(* Logix 5000 project; controller STAT 1756-L72 rev 20.12; software revision 20.04; part 20 of 34 *)
(* tags used below, declared in another part *)
   B14 : DINT[30];
   B17 : DINT[30];
   B3 : DINT[256];
   B9 : DINT[40];
   F8 : REAL[256];
   I19_000_Bit08 : ALIAS FOR I19[0].8;   // LACK DETECTIE NAOH
   I1_009_Bit03 : ALIAS FOR I1[9].3;   // Thermische storing pomp 1
   I1_009_Bit04 : ALIAS FOR I1[9].4;   // Pomp 1 in lijn
   I1_009_Bit07 : ALIAS FOR I1[9].7;   // Thermische storing pomp 2
   I1_009_Bit08 : ALIAS FOR I1[9].8;   // Pomp 2 in lijn
   I1_009_Bit09 : ALIAS FOR I1[9].9;   // Pomp 2 in driehoek
   I3_001_Bit15 : ALIAS FOR I3[1].15;   // Thermische storing voedingspomp fabriek 1
   I4_000_Bit00 : ALIAS FOR I4[0].0;   // Motor P3 voedingspomp in lijn
   I4_000_Bit03 : ALIAS FOR I4[0].3;   // Thermische storing voedingspomp fabriek 2
   I4_000_Bit04 : ALIAS FOR I4[0].4;   // Motor p4 in lijn in
   I6_000_Bit12 : ALIAS FOR I6[0].12;   // pressostaat osmose3
   N12 : DINT[230];
   N13 : DINT[230];
   N26 : DINT[256];
   N7 : DINT[255];
   O15_000_Bit04 : ALIAS FOR O15[0].4;   // RO3_EV1 RO3_EV1
   O15_000_Bit05 : ALIAS FOR O15[0].5;   // RO3_EV2 RO3_EV2
   T4 : TIMER[200];
(* ibt, continued *)

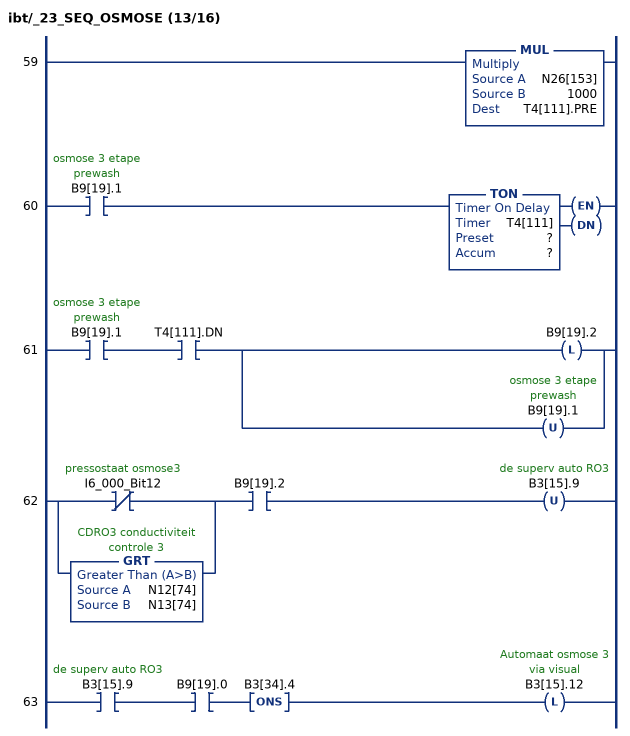
   [picture p367: ibt/_23_SEQ_OSMOSE rungs 59-63]
   59: MUL(N26[153],1000,T4[111].PRE);
   60: XIC(B9[19].1)TON(T4[111],?,?);
   61: XIC(B9[19].1)XIC(T4[111].DN)[OTL(B9[19].2) ,OTU(B9[19].1) ];
   62: [XIO(I6_000_Bit12) ,GRT(N12[74],N13[74]) ]XIC(B9[19].2)OTU(B3[15].9);
   63: XIC(B3[15].9)XIC(B9[19].0)ONS(B3[34].4)OTL(B3[15].12);
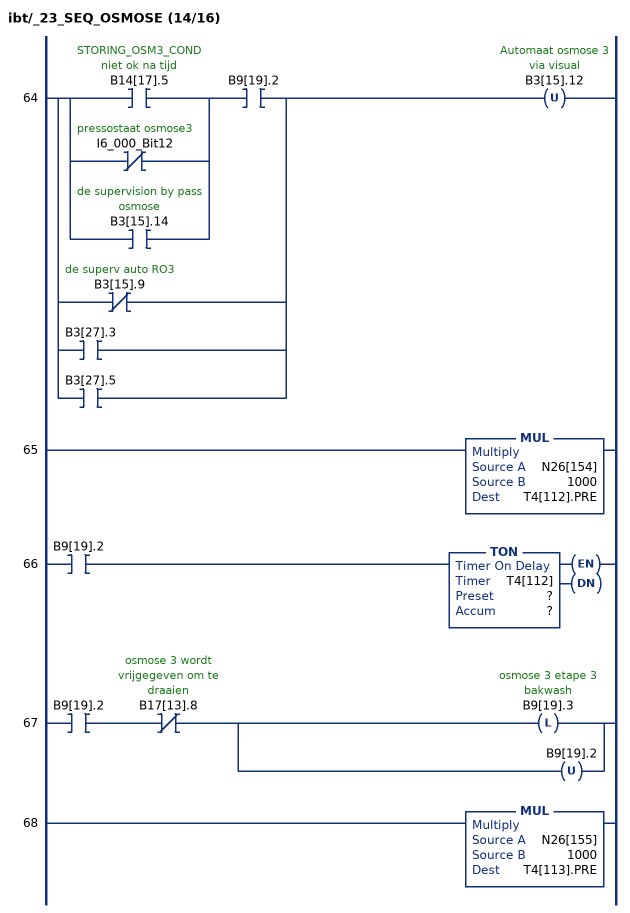
   64: [[XIC(B14[17].5) ,[XIO(I6_000_Bit12) ,XIC(B3[15].14) ] ] XIC(B9[19].2) ,XIO(B3[15].9) ,XIC(B3[27].3) ,XIC(B3[27].5) ]OTU(B3[15].12);
   65: MUL(N26[154],1000,T4[112].PRE);
   66: XIC(B9[19].2)TON(T4[112],?,?);
   67: XIC(B9[19].2)XIO(B17[13].8)[OTL(B9[19].3) ,OTU(B9[19].2) ];
   68: MUL(N26[155],1000,T4[113].PRE);
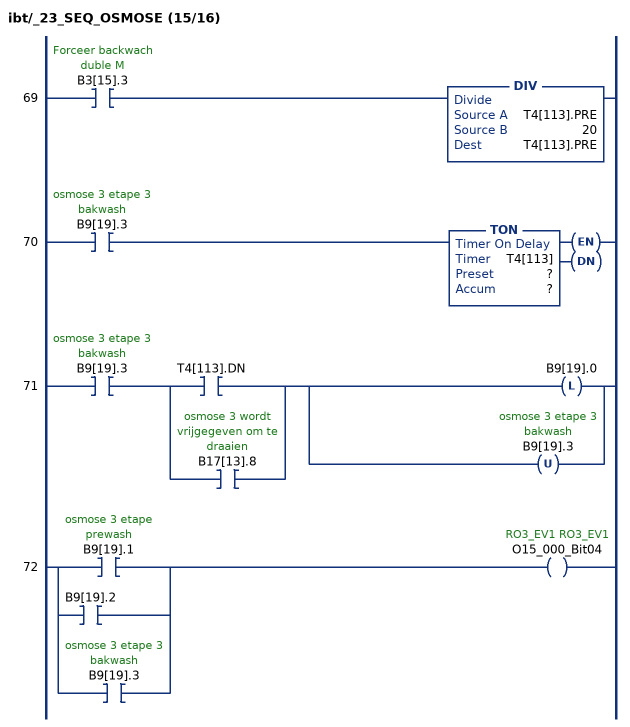
   69: XIC(B3[15].3)DIV(T4[113].PRE,20,T4[113].PRE);
   70: XIC(B9[19].3)TON(T4[113],?,?);
   71: XIC(B9[19].3)[XIC(T4[113].DN) ,XIC(B17[13].8) ][OTL(B9[19].0) ,OTU(B9[19].3) ];
   72: [XIC(B9[19].1) ,[XIC(B9[19].2) ,XIC(B9[19].3) ] ]OTE(O15_000_Bit04);
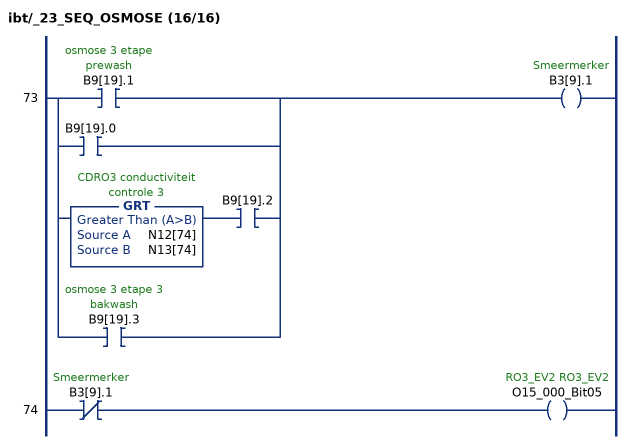
   73: [[XIC(B9[19].1) ,XIC(B9[19].0) ] ,[GRT(N12[74],N13[74]) XIC(B9[19].2) ,XIC(B9[19].3) ] ]OTE(B3[9].1);
   74: XIO(B3[9].1)OTE(O15_000_Bit05);
END_ROUTINE

ROUTINE _24_ALARMING   (* ladder *)
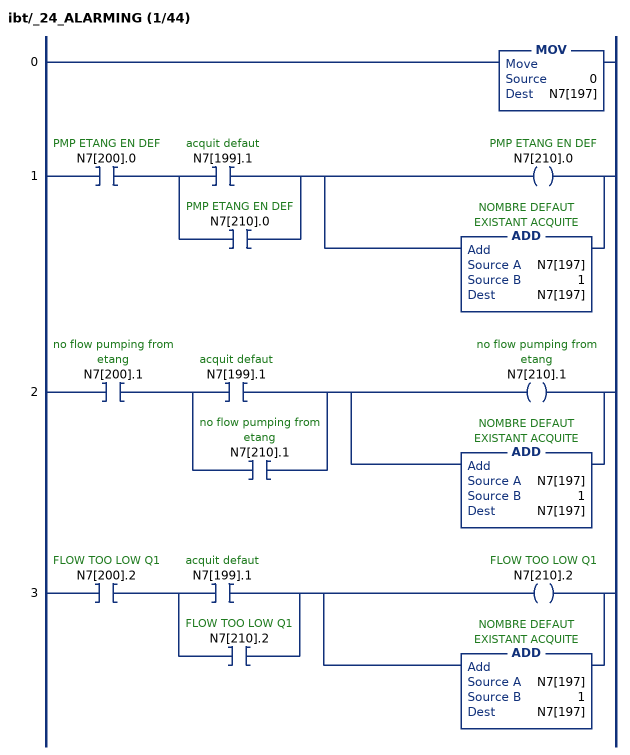
   0: MOV(0,N7[197]);
   1: XIC(N7[200].0)[XIC(N7[199].1) ,XIC(N7[210].0) ][OTE(N7[210].0) ,ADD(N7[197],1,N7[197]) ];
   2: XIC(N7[200].1)[XIC(N7[199].1) ,XIC(N7[210].1) ][OTE(N7[210].1) ,ADD(N7[197],1,N7[197]) ];
   3: XIC(N7[200].2)[XIC(N7[199].1) ,XIC(N7[210].2) ][OTE(N7[210].2) ,ADD(N7[197],1,N7[197]) ];
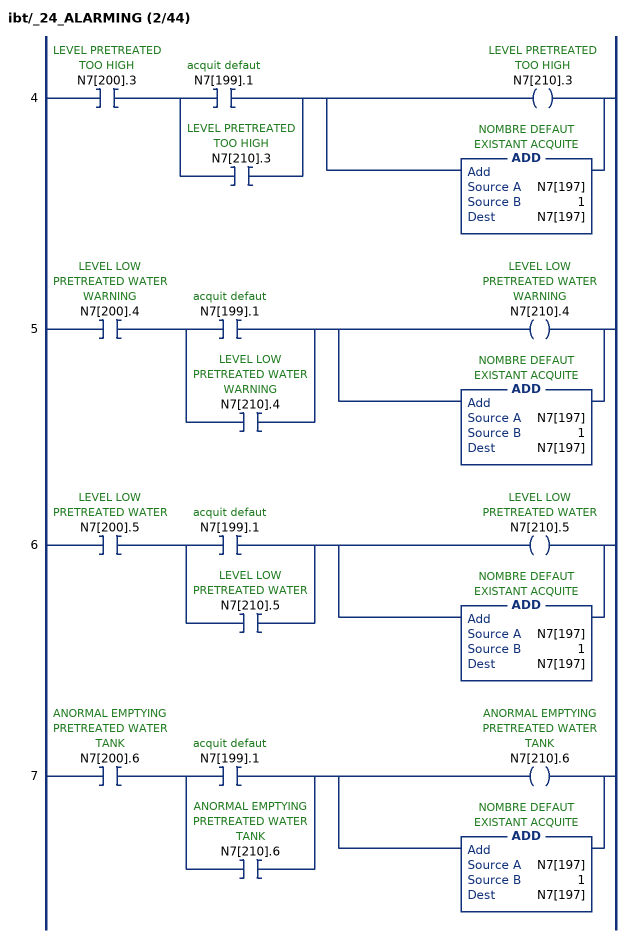
   4: XIC(N7[200].3)[XIC(N7[199].1) ,XIC(N7[210].3) ][OTE(N7[210].3) ,ADD(N7[197],1,N7[197]) ];
   5: XIC(N7[200].4)[XIC(N7[199].1) ,XIC(N7[210].4) ][OTE(N7[210].4) ,ADD(N7[197],1,N7[197]) ];
   6: XIC(N7[200].5)[XIC(N7[199].1) ,XIC(N7[210].5) ][OTE(N7[210].5) ,ADD(N7[197],1,N7[197]) ];
   7: XIC(N7[200].6)[XIC(N7[199].1) ,XIC(N7[210].6) ][OTE(N7[210].6) ,ADD(N7[197],1,N7[197]) ];
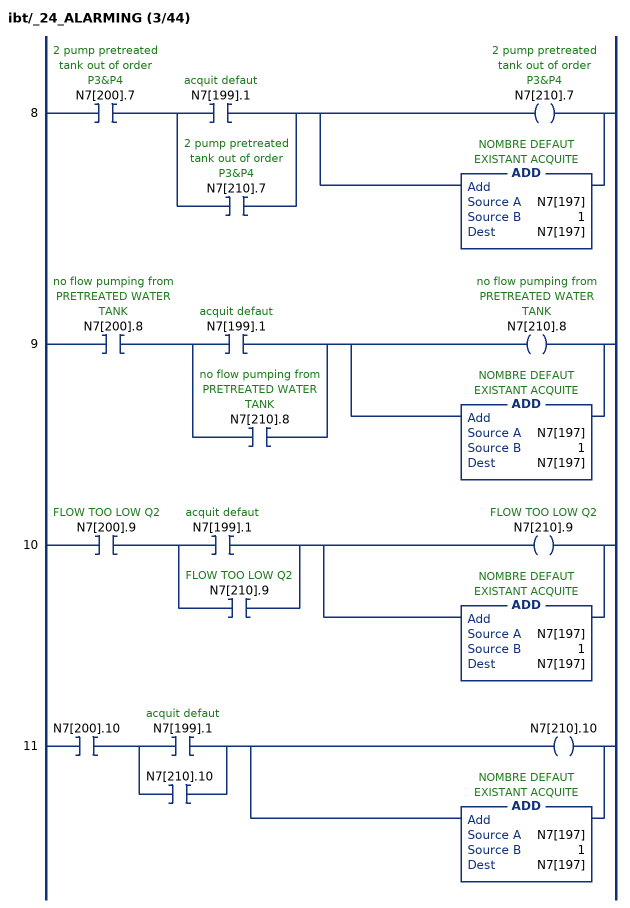
   8: XIC(N7[200].7)[XIC(N7[199].1) ,XIC(N7[210].7) ][OTE(N7[210].7) ,ADD(N7[197],1,N7[197]) ];
   9: XIC(N7[200].8)[XIC(N7[199].1) ,XIC(N7[210].8) ][OTE(N7[210].8) ,ADD(N7[197],1,N7[197]) ];
   10: XIC(N7[200].9)[XIC(N7[199].1) ,XIC(N7[210].9) ][OTE(N7[210].9) ,ADD(N7[197],1,N7[197]) ];
   11: XIC(N7[200].10)[XIC(N7[199].1) ,XIC(N7[210].10) ][OTE(N7[210].10) ,ADD(N7[197],1,N7[197]) ];
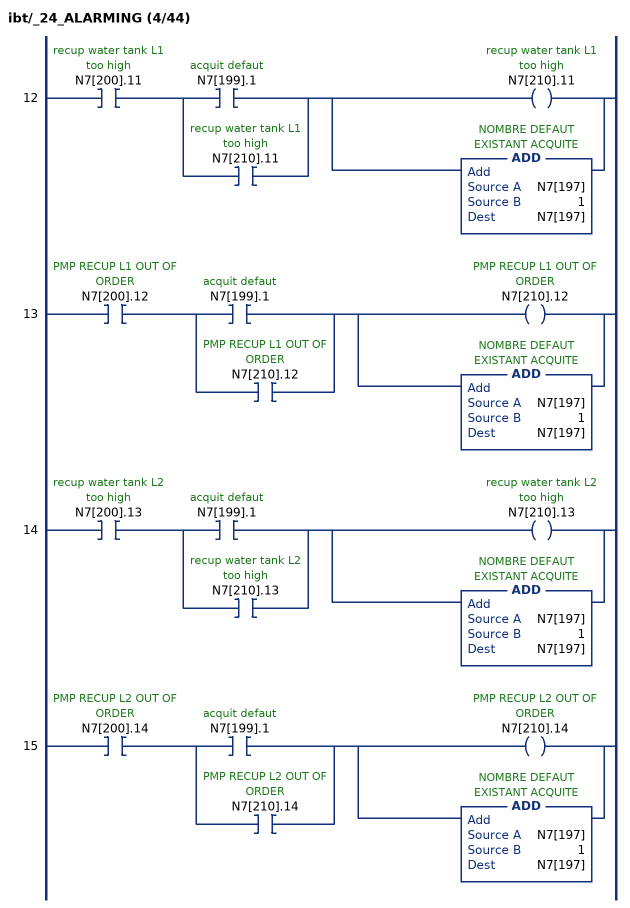
   12: XIC(N7[200].11)[XIC(N7[199].1) ,XIC(N7[210].11) ][OTE(N7[210].11) ,ADD(N7[197],1,N7[197]) ];
   13: XIC(N7[200].12)[XIC(N7[199].1) ,XIC(N7[210].12) ][OTE(N7[210].12) ,ADD(N7[197],1,N7[197]) ];
   14: XIC(N7[200].13)[XIC(N7[199].1) ,XIC(N7[210].13) ][OTE(N7[210].13) ,ADD(N7[197],1,N7[197]) ];
   15: XIC(N7[200].14)[XIC(N7[199].1) ,XIC(N7[210].14) ][OTE(N7[210].14) ,ADD(N7[197],1,N7[197]) ];
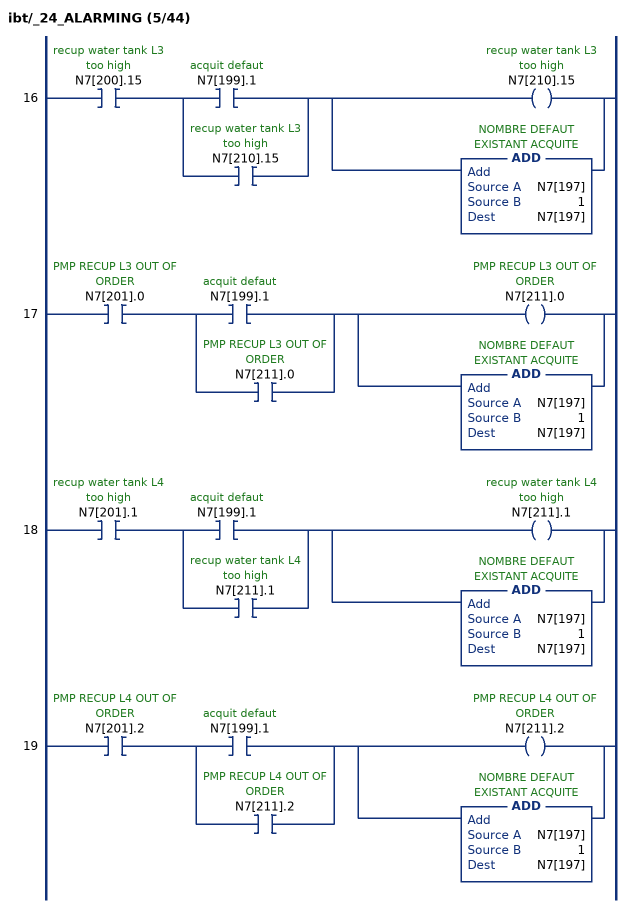
   16: XIC(N7[200].15)[XIC(N7[199].1) ,XIC(N7[210].15) ][OTE(N7[210].15) ,ADD(N7[197],1,N7[197]) ];
   17: XIC(N7[201].0)[XIC(N7[199].1) ,XIC(N7[211].0) ][OTE(N7[211].0) ,ADD(N7[197],1,N7[197]) ];
   18: XIC(N7[201].1)[XIC(N7[199].1) ,XIC(N7[211].1) ][OTE(N7[211].1) ,ADD(N7[197],1,N7[197]) ];
   19: XIC(N7[201].2)[XIC(N7[199].1) ,XIC(N7[211].2) ][OTE(N7[211].2) ,ADD(N7[197],1,N7[197]) ];
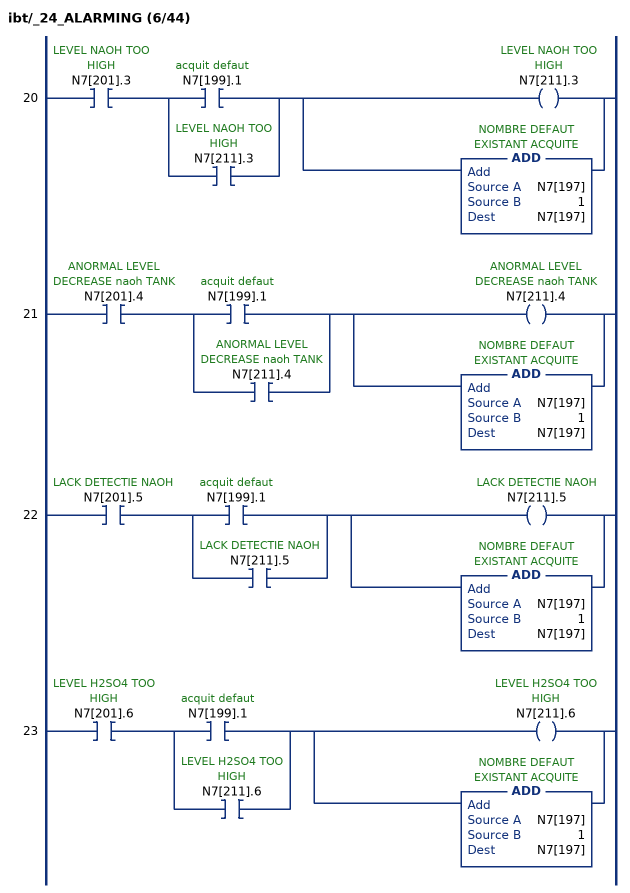
   20: XIC(N7[201].3)[XIC(N7[199].1) ,XIC(N7[211].3) ][OTE(N7[211].3) ,ADD(N7[197],1,N7[197]) ];
   21: XIC(N7[201].4)[XIC(N7[199].1) ,XIC(N7[211].4) ][OTE(N7[211].4) ,ADD(N7[197],1,N7[197]) ];
   22: XIC(N7[201].5)[XIC(N7[199].1) ,XIC(N7[211].5) ][OTE(N7[211].5) ,ADD(N7[197],1,N7[197]) ];
   23: XIC(N7[201].6)[XIC(N7[199].1) ,XIC(N7[211].6) ][OTE(N7[211].6) ,ADD(N7[197],1,N7[197]) ];
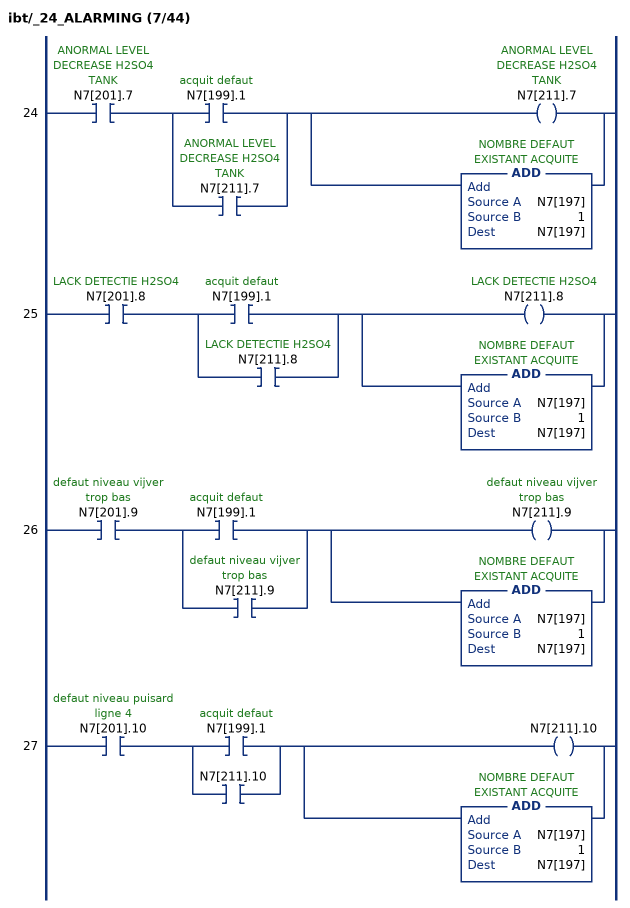
   24: XIC(N7[201].7)[XIC(N7[199].1) ,XIC(N7[211].7) ][OTE(N7[211].7) ,ADD(N7[197],1,N7[197]) ];
   25: XIC(N7[201].8)[XIC(N7[199].1) ,XIC(N7[211].8) ][OTE(N7[211].8) ,ADD(N7[197],1,N7[197]) ];
   26: XIC(N7[201].9)[XIC(N7[199].1) ,XIC(N7[211].9) ][OTE(N7[211].9) ,ADD(N7[197],1,N7[197]) ];
   27: XIC(N7[201].10)[XIC(N7[199].1) ,XIC(N7[211].10) ][OTE(N7[211].10) ,ADD(N7[197],1,N7[197]) ];
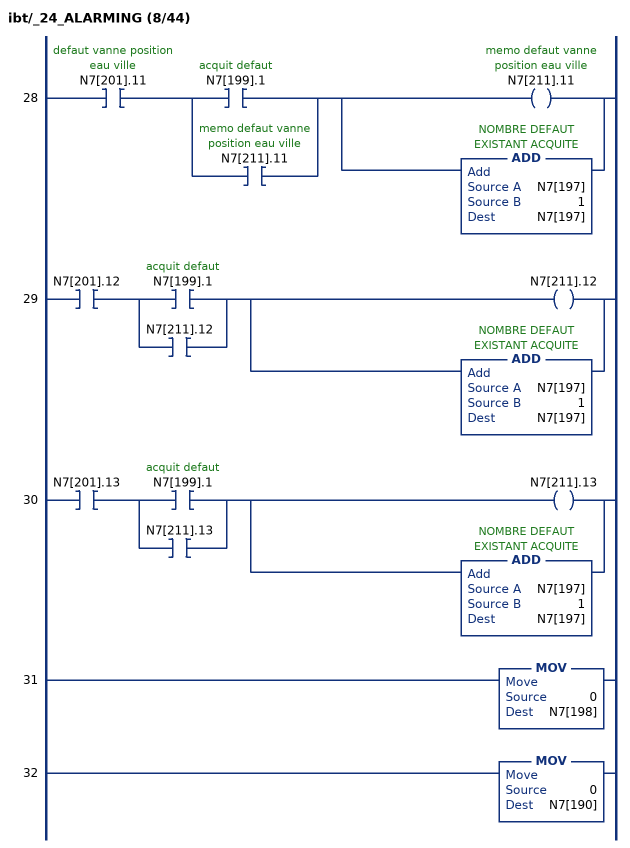
   28: XIC(N7[201].11)[XIC(N7[199].1) ,XIC(N7[211].11) ][OTE(N7[211].11) ,ADD(N7[197],1,N7[197]) ];
   29: XIC(N7[201].12)[XIC(N7[199].1) ,XIC(N7[211].12) ][OTE(N7[211].12) ,ADD(N7[197],1,N7[197]) ];
   30: XIC(N7[201].13)[XIC(N7[199].1) ,XIC(N7[211].13) ][OTE(N7[211].13) ,ADD(N7[197],1,N7[197]) ];
   31: MOV(0,N7[198]);
   32: MOV(0,N7[190]);
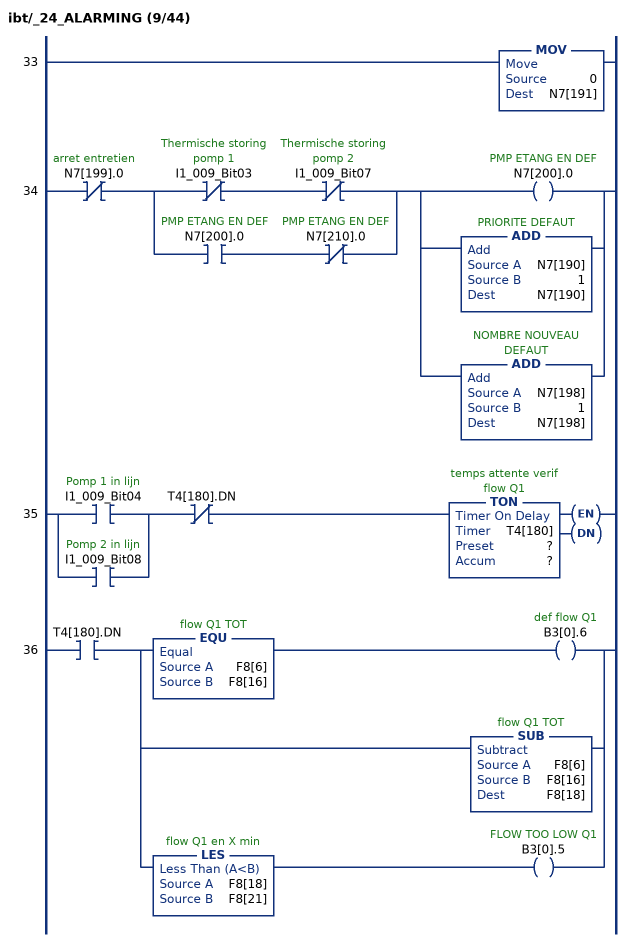
   33: MOV(0,N7[191]);
   34: XIO(N7[199].0)[XIO(I1_009_Bit03) XIO(I1_009_Bit07) ,XIC(N7[200].0) XIO(N7[210].0) ][OTE(N7[200].0) ,ADD(N7[190],1,N7[190]) ,ADD(N7[198],1,N7[198]) ];
   35: [XIC(I1_009_Bit04) ,XIC(I1_009_Bit08) ]XIO(T4[180].DN)TON(T4[180],?,?);
   36: XIC(T4[180].DN)[EQU(F8[6],F8[16]) OTE(B3[0].6) ,SUB(F8[6],F8[16],F8[18]) ,LES(F8[18],F8[21]) OTE(B3[0].5) ];
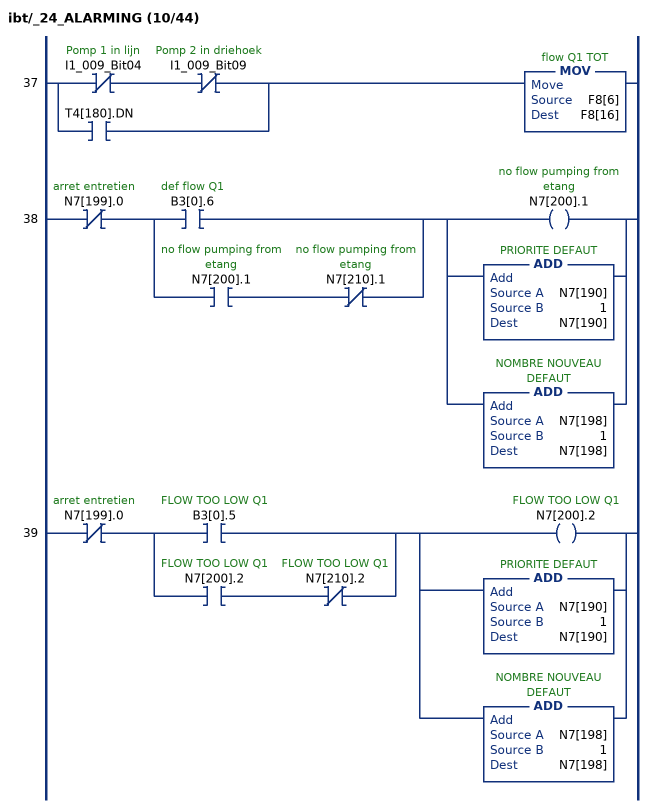
   37: [XIO(I1_009_Bit04) XIO(I1_009_Bit09) ,XIC(T4[180].DN) ]MOV(F8[6],F8[16]);
   38: XIO(N7[199].0)[XIC(B3[0].6) ,XIC(N7[200].1) XIO(N7[210].1) ][OTE(N7[200].1) ,ADD(N7[190],1,N7[190]) ,ADD(N7[198],1,N7[198]) ];
   39: XIO(N7[199].0)[XIC(B3[0].5) ,XIC(N7[200].2) XIO(N7[210].2) ][OTE(N7[200].2) ,ADD(N7[190],1,N7[190]) ,ADD(N7[198],1,N7[198]) ];
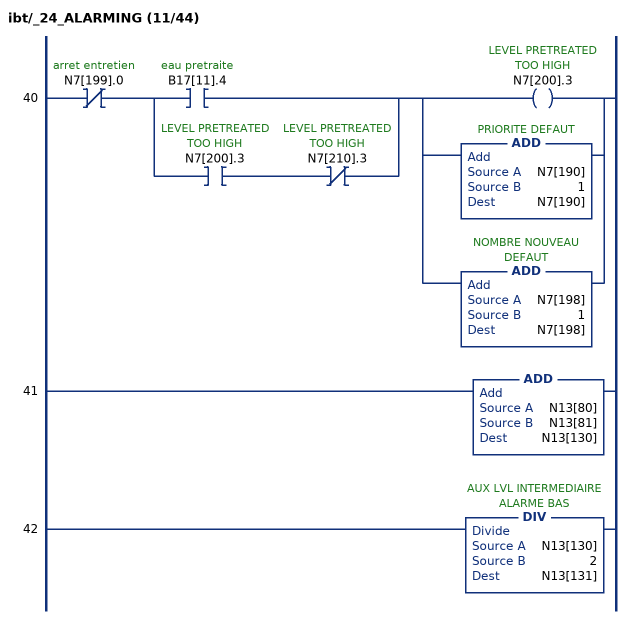
   40: XIO(N7[199].0)[XIC(B17[11].4) ,XIC(N7[200].3) XIO(N7[210].3) ][OTE(N7[200].3) ,ADD(N7[190],1,N7[190]) ,ADD(N7[198],1,N7[198]) ];
   41: ADD(N13[80],N13[81],N13[130]);
   42: DIV(N13[130],2,N13[131]);
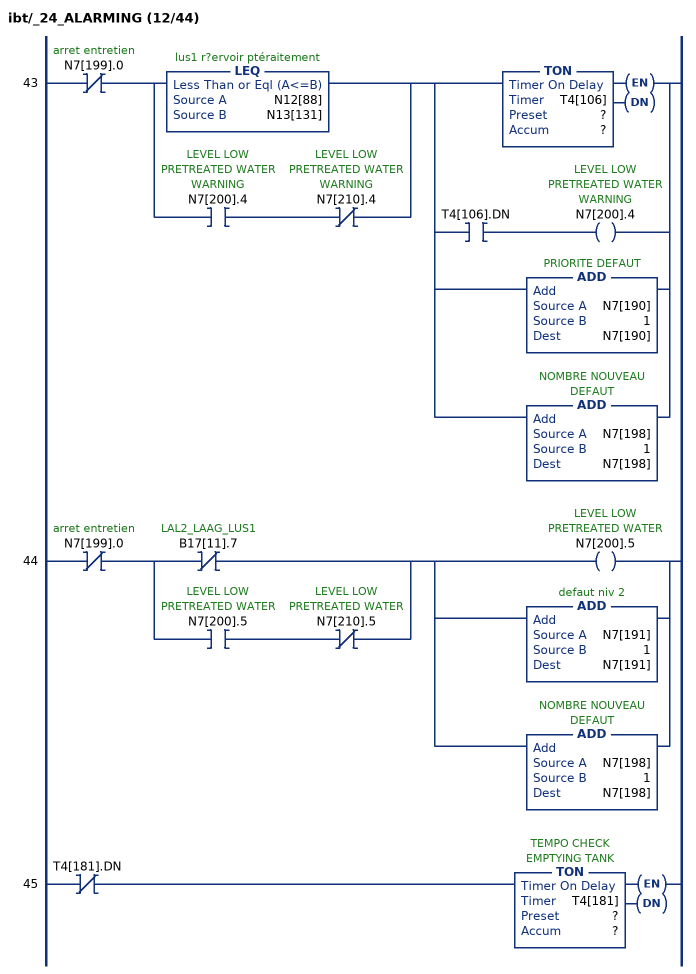
   43: XIO(N7[199].0)[LEQ(N12[88],N13[131]) ,XIC(N7[200].4) XIO(N7[210].4) ][TON(T4[106],?,?) ,XIC(T4[106].DN) OTE(N7[200].4) ,ADD(N7[190],1,N7[190]) ,ADD(N7[198],1,N7[198]) ];
   44: XIO(N7[199].0)[XIO(B17[11].7) ,XIC(N7[200].5) XIO(N7[210].5) ][OTE(N7[200].5) ,ADD(N7[191],1,N7[191]) ,ADD(N7[198],1,N7[198]) ];
   45: XIO(T4[181].DN)TON(T4[181],?,?);
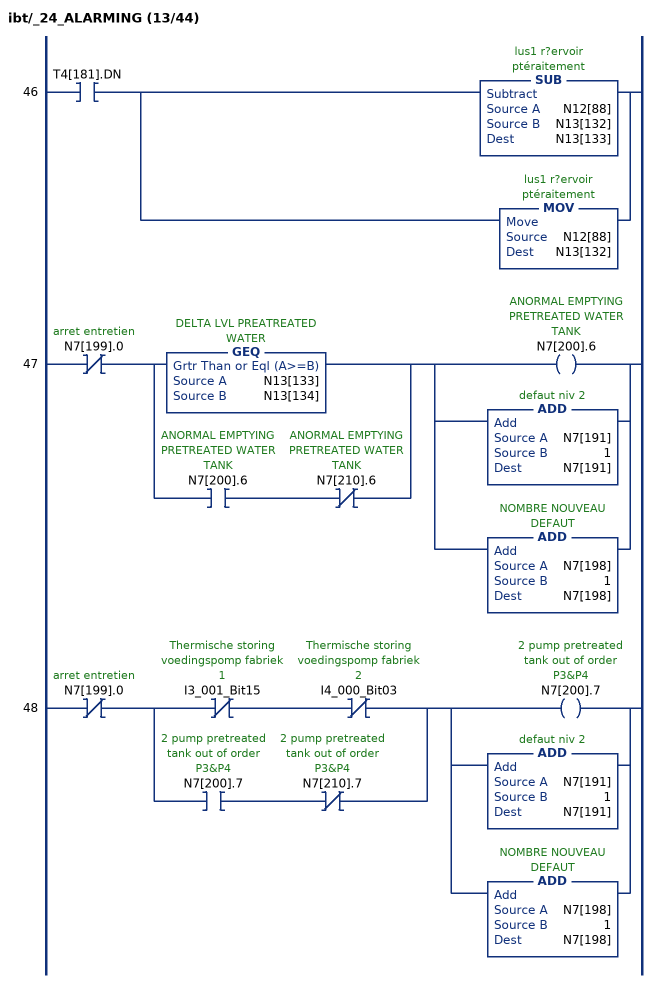
   46: XIC(T4[181].DN)[SUB(N12[88],N13[132],N13[133]) ,MOV(N12[88],N13[132]) ];
   47: XIO(N7[199].0)[GEQ(N13[133],N13[134]) ,XIC(N7[200].6) XIO(N7[210].6) ][OTE(N7[200].6) ,ADD(N7[191],1,N7[191]) ,ADD(N7[198],1,N7[198]) ];
   48: XIO(N7[199].0)[XIO(I3_001_Bit15) XIO(I4_000_Bit03) ,XIC(N7[200].7) XIO(N7[210].7) ][OTE(N7[200].7) ,ADD(N7[191],1,N7[191]) ,ADD(N7[198],1,N7[198]) ];
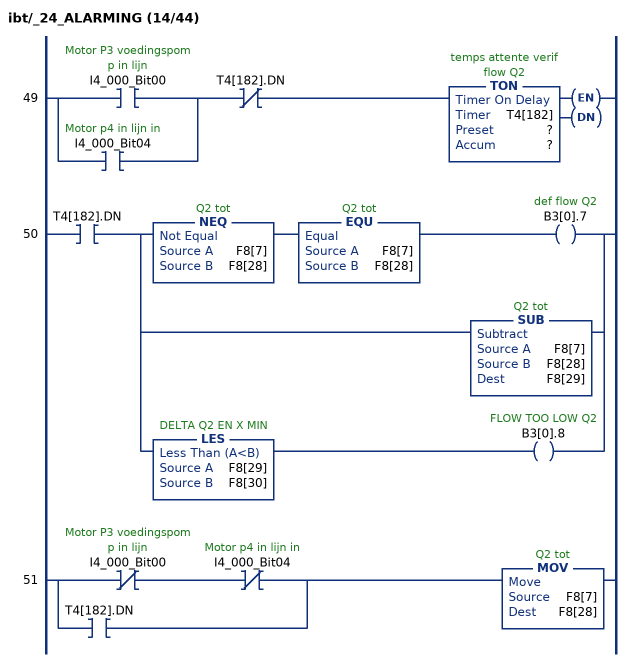
   49: [XIC(I4_000_Bit00) ,XIC(I4_000_Bit04) ]XIO(T4[182].DN)TON(T4[182],?,?);
   50: XIC(T4[182].DN)[NEQ(F8[7],F8[28]) EQU(F8[7],F8[28]) OTE(B3[0].7) ,SUB(F8[7],F8[28],F8[29]) ,LES(F8[29],F8[30]) OTE(B3[0].8) ];
   51: [XIO(I4_000_Bit00) XIO(I4_000_Bit04) ,XIC(T4[182].DN) ]MOV(F8[7],F8[28]);
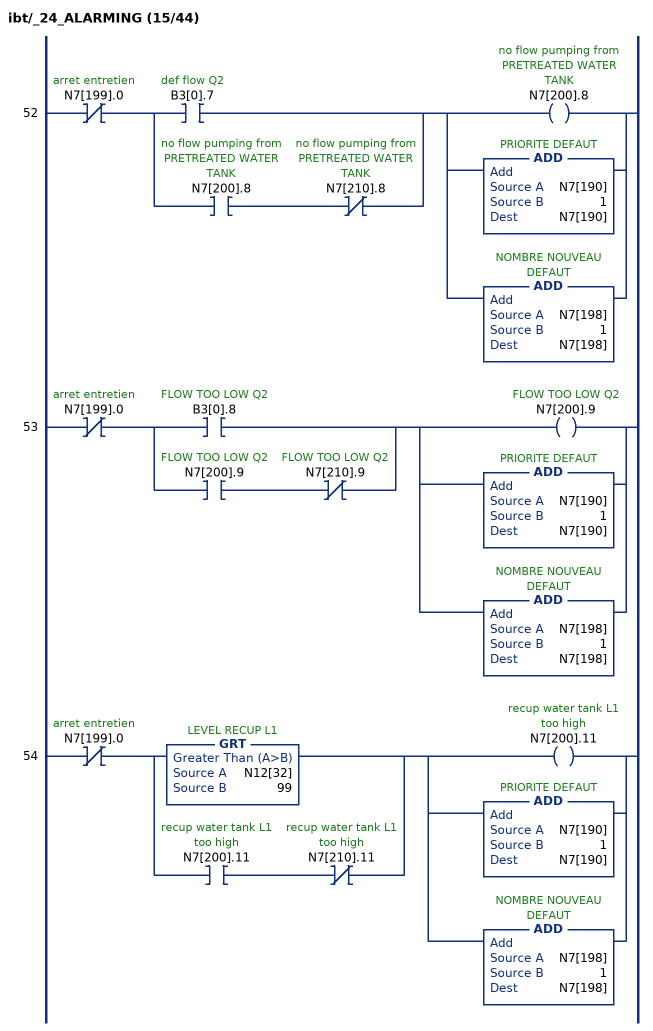
   52: XIO(N7[199].0)[XIC(B3[0].7) ,XIC(N7[200].8) XIO(N7[210].8) ][OTE(N7[200].8) ,ADD(N7[190],1,N7[190]) ,ADD(N7[198],1,N7[198]) ];
   53: XIO(N7[199].0)[XIC(B3[0].8) ,XIC(N7[200].9) XIO(N7[210].9) ][OTE(N7[200].9) ,ADD(N7[190],1,N7[190]) ,ADD(N7[198],1,N7[198]) ];
   54: XIO(N7[199].0)[GRT(N12[32],99) ,XIC(N7[200].11) XIO(N7[210].11) ][OTE(N7[200].11) ,ADD(N7[190],1,N7[190]) ,ADD(N7[198],1,N7[198]) ];
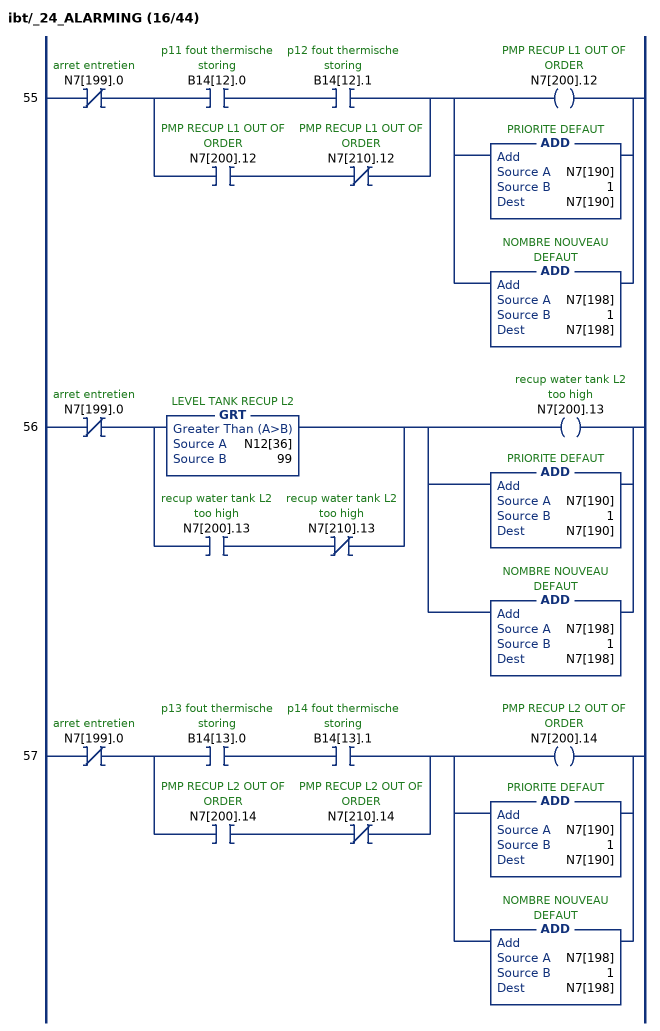
   55: XIO(N7[199].0)[XIC(B14[12].0) XIC(B14[12].1) ,XIC(N7[200].12) XIO(N7[210].12) ][OTE(N7[200].12) ,ADD(N7[190],1,N7[190]) ,ADD(N7[198],1,N7[198]) ];
   56: XIO(N7[199].0)[GRT(N12[36],99) ,XIC(N7[200].13) XIO(N7[210].13) ][OTE(N7[200].13) ,ADD(N7[190],1,N7[190]) ,ADD(N7[198],1,N7[198]) ];
   57: XIO(N7[199].0)[XIC(B14[13].0) XIC(B14[13].1) ,XIC(N7[200].14) XIO(N7[210].14) ][OTE(N7[200].14) ,ADD(N7[190],1,N7[190]) ,ADD(N7[198],1,N7[198]) ];
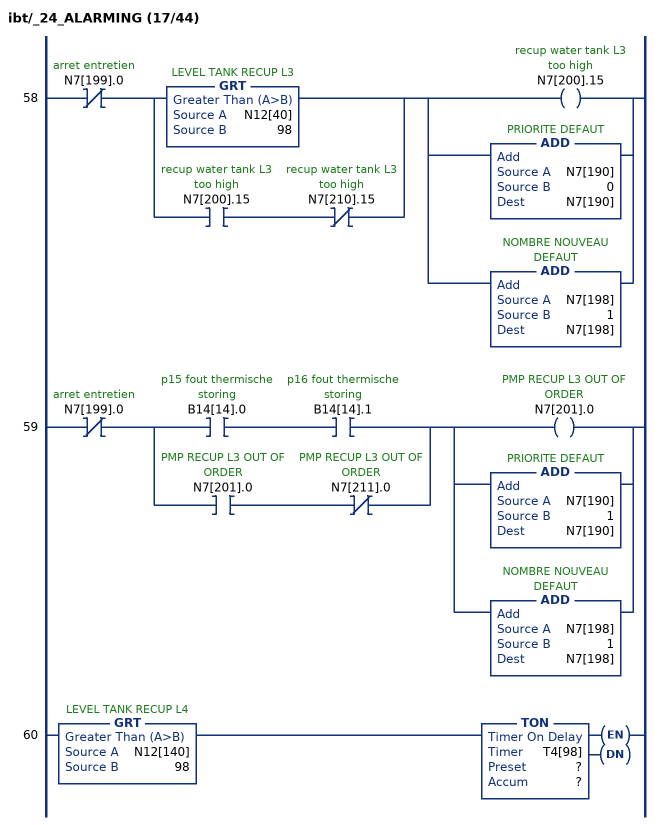
   58: XIO(N7[199].0)[GRT(N12[40],98) ,XIC(N7[200].15) XIO(N7[210].15) ][OTE(N7[200].15) ,ADD(N7[190],0,N7[190]) ,ADD(N7[198],1,N7[198]) ];
   59: XIO(N7[199].0)[XIC(B14[14].0) XIC(B14[14].1) ,XIC(N7[201].0) XIO(N7[211].0) ][OTE(N7[201].0) ,ADD(N7[190],1,N7[190]) ,ADD(N7[198],1,N7[198]) ];
   60: GRT(N12[140],98)TON(T4[98],?,?);
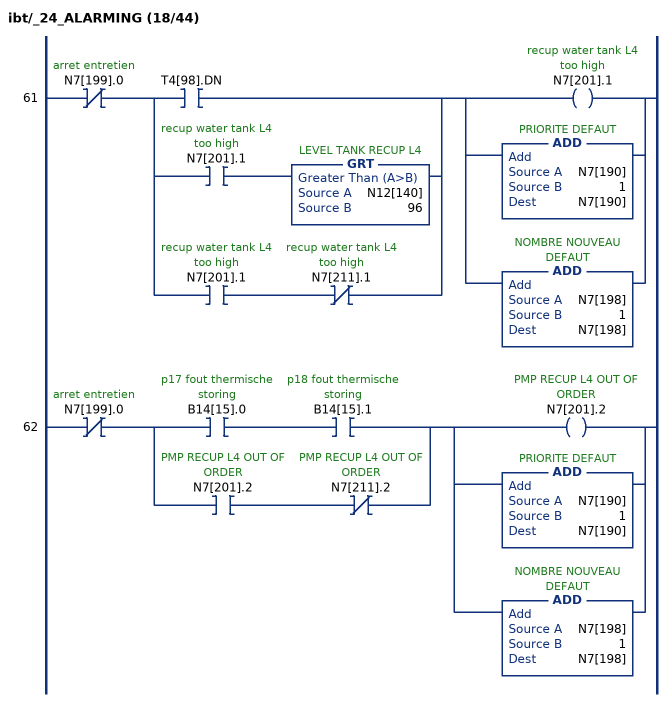
   61: XIO(N7[199].0)[[XIC(T4[98].DN) ,XIC(N7[201].1) GRT(N12[140],96) ] ,XIC(N7[201].1) XIO(N7[211].1) ][OTE(N7[201].1) ,ADD(N7[190],1,N7[190]) ,ADD(N7[198],1,N7[198]) ];
   62: XIO(N7[199].0)[XIC(B14[15].0) XIC(B14[15].1) ,XIC(N7[201].2) XIO(N7[211].2) ][OTE(N7[201].2) ,ADD(N7[190],1,N7[190]) ,ADD(N7[198],1,N7[198]) ];
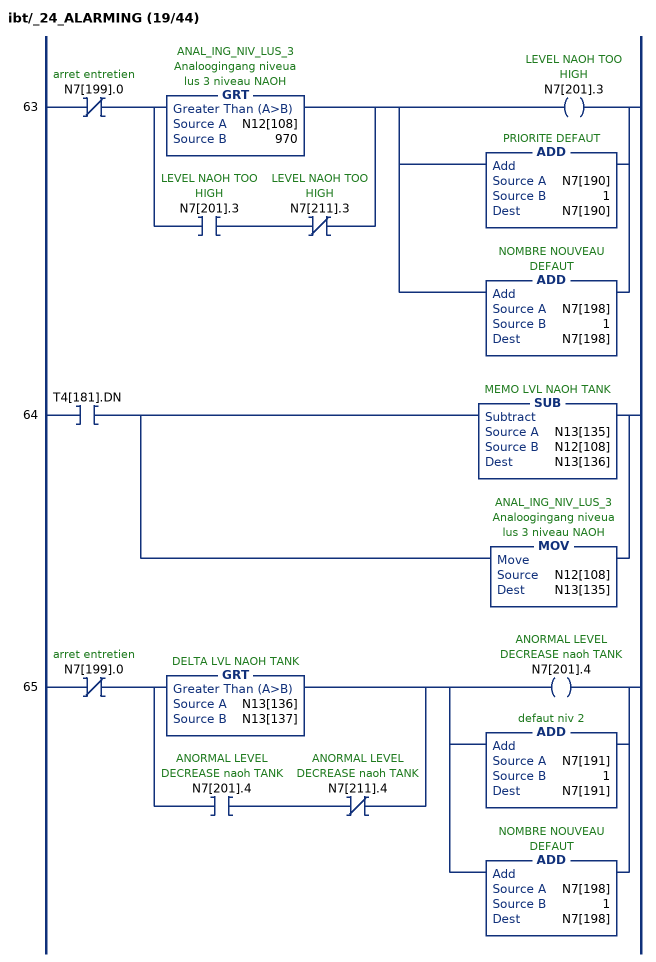
   63: XIO(N7[199].0)[GRT(N12[108],970) ,XIC(N7[201].3) XIO(N7[211].3) ][OTE(N7[201].3) ,ADD(N7[190],1,N7[190]) ,ADD(N7[198],1,N7[198]) ];
   64: XIC(T4[181].DN)[SUB(N13[135],N12[108],N13[136]) ,MOV(N12[108],N13[135]) ];
   65: XIO(N7[199].0)[GRT(N13[136],N13[137]) ,XIC(N7[201].4) XIO(N7[211].4) ][OTE(N7[201].4) ,ADD(N7[191],1,N7[191]) ,ADD(N7[198],1,N7[198]) ];
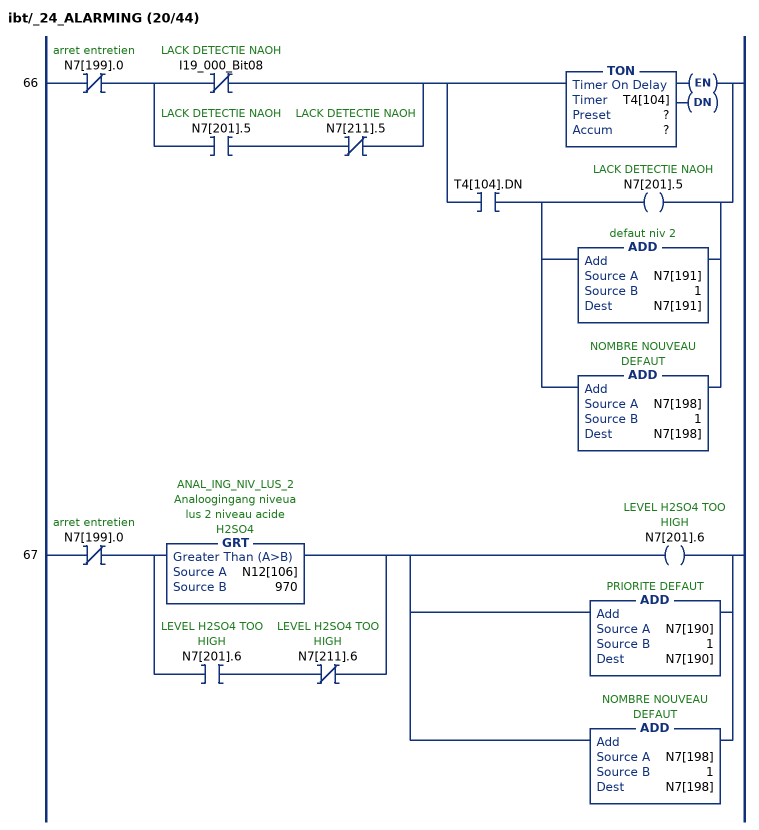
   66: XIO(N7[199].0)[XIO(I19_000_Bit08) ,XIC(N7[201].5) XIO(N7[211].5) ][TON(T4[104],?,?) ,XIC(T4[104].DN) [OTE(N7[201].5) ,ADD(N7[191],1,N7[191]) ,ADD(N7[198],1,N7[198]) ] ];
   67: XIO(N7[199].0)[GRT(N12[106],970) ,XIC(N7[201].6) XIO(N7[211].6) ][OTE(N7[201].6) ,ADD(N7[190],1,N7[190]) ,ADD(N7[198],1,N7[198]) ];
